TYPE ST_SettingsTransportLift :
STRUCT
	//Lift
	stLiftSpeedProfileJogging : ST_SpeedProfile;
	stLiftSpeedProfilePositioning : ST_SpeedProfile;   
	arr_LiftPositioningProfile : ARRAY[0..10] OF ST_PositioningProfile;
	
	//Transport Unit
	stTransportUintSpeedProfileJogging : ST_SpeedProfile;
	stTransportSpeedProfilePositioning : ST_SpeedProfile;
	arr_TransportUnitPositioningProfile : ARRAY[0..5] OF ST_PositioningProfile;
	
	//--stLiftIdle : ST_PositioningProfile;
	
	//--stLiftPrePickTrolleyInTB : ST_PositioningProfile; 
	//--stLiftPickTrolleyInTB : ST_PositioningProfile;
	//--stLiftRaiseTrolleyInTB : ST_PositioningProfile;
	
	//--stLiftPrePlaceTrolleyInCabin : ST_PositioningProfile;
	//--stLiftPlaceTrolleyInCabin : ST_PositioningProfile;
	//--stLiftPrePickTrolleyInCabin : ST_PositioningProfile;
	//--stLiftPickTrolleyInCabin : ST_PositioningProfile;

	//--stLiftRaiseTrolleyInCabin : ST_PositioningProfile;
	//--stLiftPrePlaceTrolleyInTB : ST_PositioningProfile;
	//--stLiftPlaceTrolleyInTB : ST_PositioningProfile;
	

END_STRUCT
END_TYPE

(* stored: Version 1.1.0.1, ProductVersion 3.1.4024.12
   DUT ST_SettingsTransportLift: Id {cad671c8-daf9-4539-9908-38693c7e494e} *)
